{attribute 'GeneratedUsingTerminal: EJ1918-0000-0017'}
{attribute addProperty BoxType "EJ1918-0000-0017"}
{attribute addProperty Id "FSoE_InputsFSoE_Inputs_C661B78A17FSoE_OutputsFSoE_Outputs_E138FCB59"}
{attribute addProperty CRC "418223391"}
{attribute addProperty Size "26"}
TYPE Module_1_FSOE_18ED951F :
STRUCT
	{attribute addProperty Name "FSoE_Inputs"}
	FSoE_Inputs  : FSoE_Inputs_C661B78A;
	{attribute addProperty Name "FSoE_Outputs"}
	FSoE_Outputs  : FSoE_Outputs_E138FCB5;
END_STRUCT
END_TYPE

(* stored: Version 1.2.0.0, ProductVersion 3.1.4024.9
   DUT Module_1_FSOE_18ED951F: Id {07490694-9334-4884-b4ed-53cc130fd559} *)
